(********************************************************************************************)
(*							Beckhoff Automation Poland										*)
(*								FB_Blink_S	 v1.1											*)
(*									9.11.2007												*)
(*						Blok funkcyjny zegara synchronicznego								*)
(*__________________________________________________________________________________________*)

FUNCTION_BLOCK FB_Blink_S
VAR_INPUT
	Tv										:	TIME;				(*Czas trwania impulsu i przerwy*)
END_VAR
VAR_OUTPUT
	Q										:	BOOL;				(*Wyjscie*)
END_VAR
VAR
	ton1									:	TON;
	ton2									:	TON;
END_VAR

ton1(IN:= NOT ton2.Q, PT:=Tv);
Q:=ton1.Q;
ton2(IN:=ton1.Q , PT:=ton1.PT );

END_FUNCTION_BLOCK

(* stored: Version 1.1.0.1, ProductVersion 3.1.4026.13, FileIdentifier fd193d9c3adb510df775a229a19aa43ceb16be11, FileSignature 047dbe3a97825e99a78edc852774312469fd9528cda607eac604233bcc888cfec6b4451006167186b82edb5cb110e8f813119c9bb30ed9d12eb03e68e2b6d64edb1d03123095f77ab509f16a19edfe5a3778524196602079b3517523eb3cc4090b69d3c519fc4bb5ee13ba6466b3e4032cb2c9a33035decc71190bc2fad8edb4e2ed2932fb61c78229ecf486e8644c9d091fd1da97a1a9fe086765e8cc30bdd4ea9c86bcb6bfa96480f717387476606a5b02b57e76f415ab7e239b24b930ac3dda0a59fba7e2a31a0ef626ed2b95a0338dfd130beefc5c82ce6c7629f3b05ca91582c4855d8eab0b469120563eedf552b2ac6032aff79d9624ae7b7d50c39d8a
   POU FB_Blink_S: Id {73ad219d-f669-44b3-a222-006b3bb133de}, SpecialFunc None *)
